{attribute 'qualified_only'}
{attribute 'strict'}
TYPE E_ServoVise_Command :
(
	NoCommand,
	Attach,
	MoveToPos,
	Release,
	Fix
);
END_TYPE

(* stored: Version 1.1.0.1, ProductVersion 3.1.4024.12
   EnumerationTextList E_ServoVise_Command: Id {b2230f0a-eb94-48ac-84a3-8206d0e0c304} *)
